# B&R Automation Studio project DuctLines (part 3)

### Program Logical/Feeder (IEC)

#### Cyclic.ld - Cyclic code
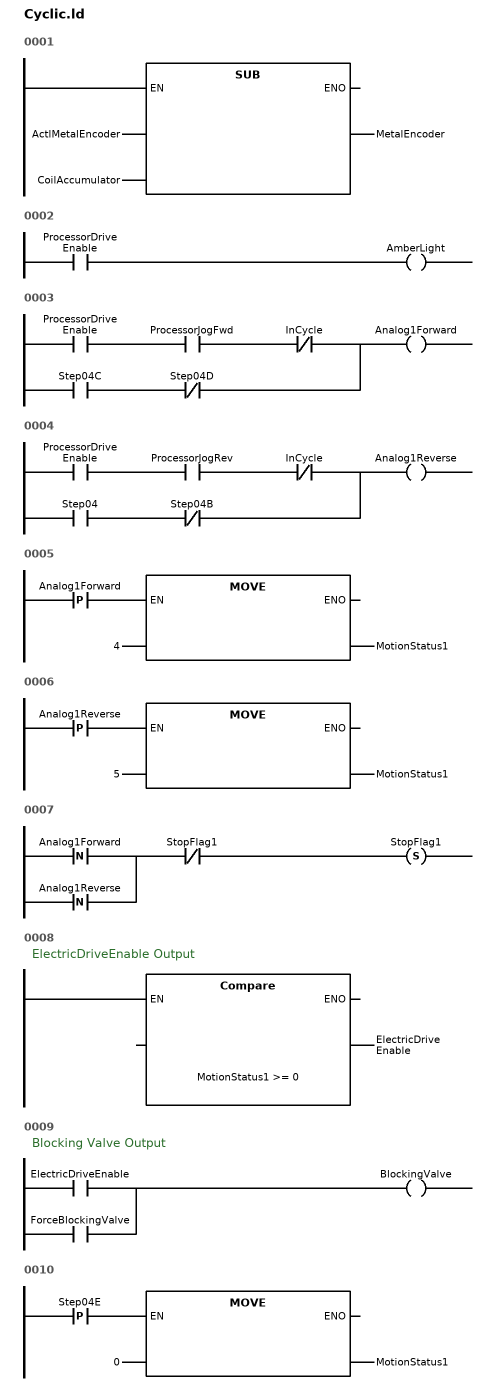
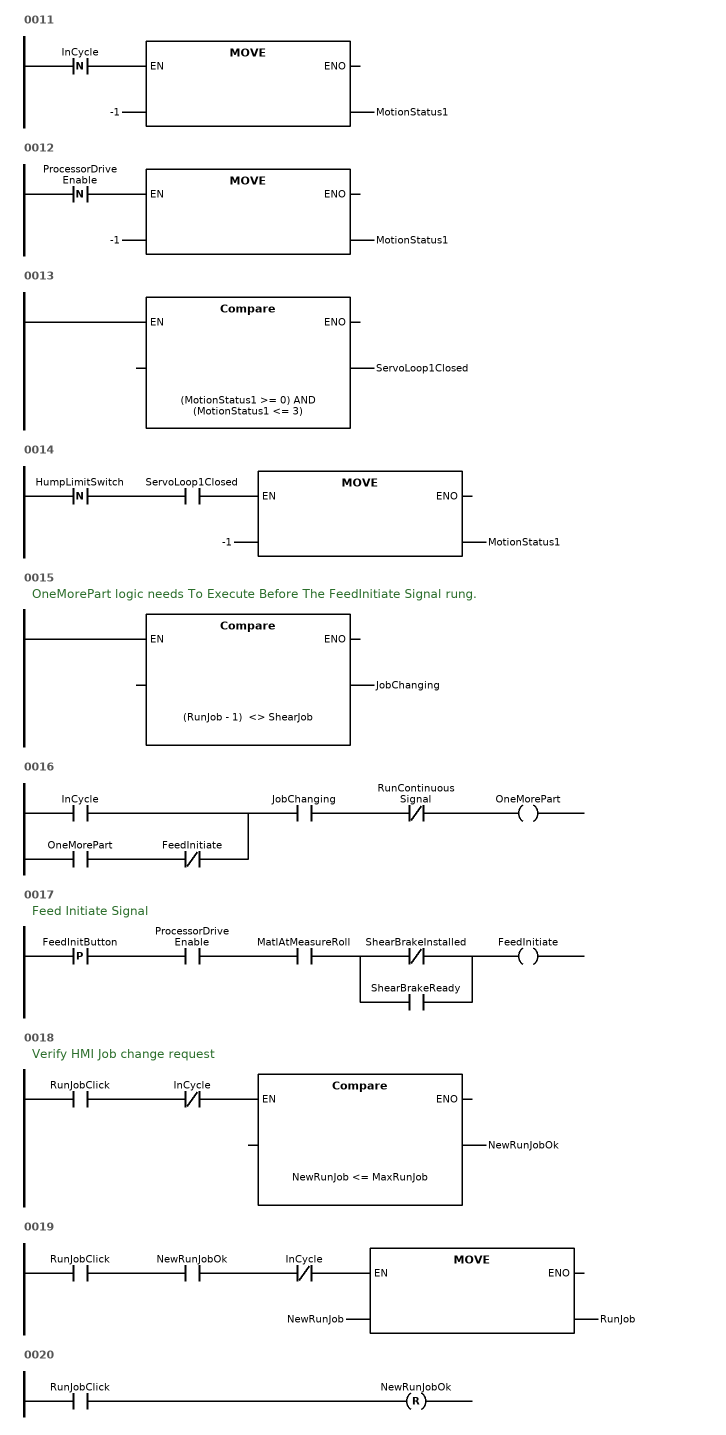
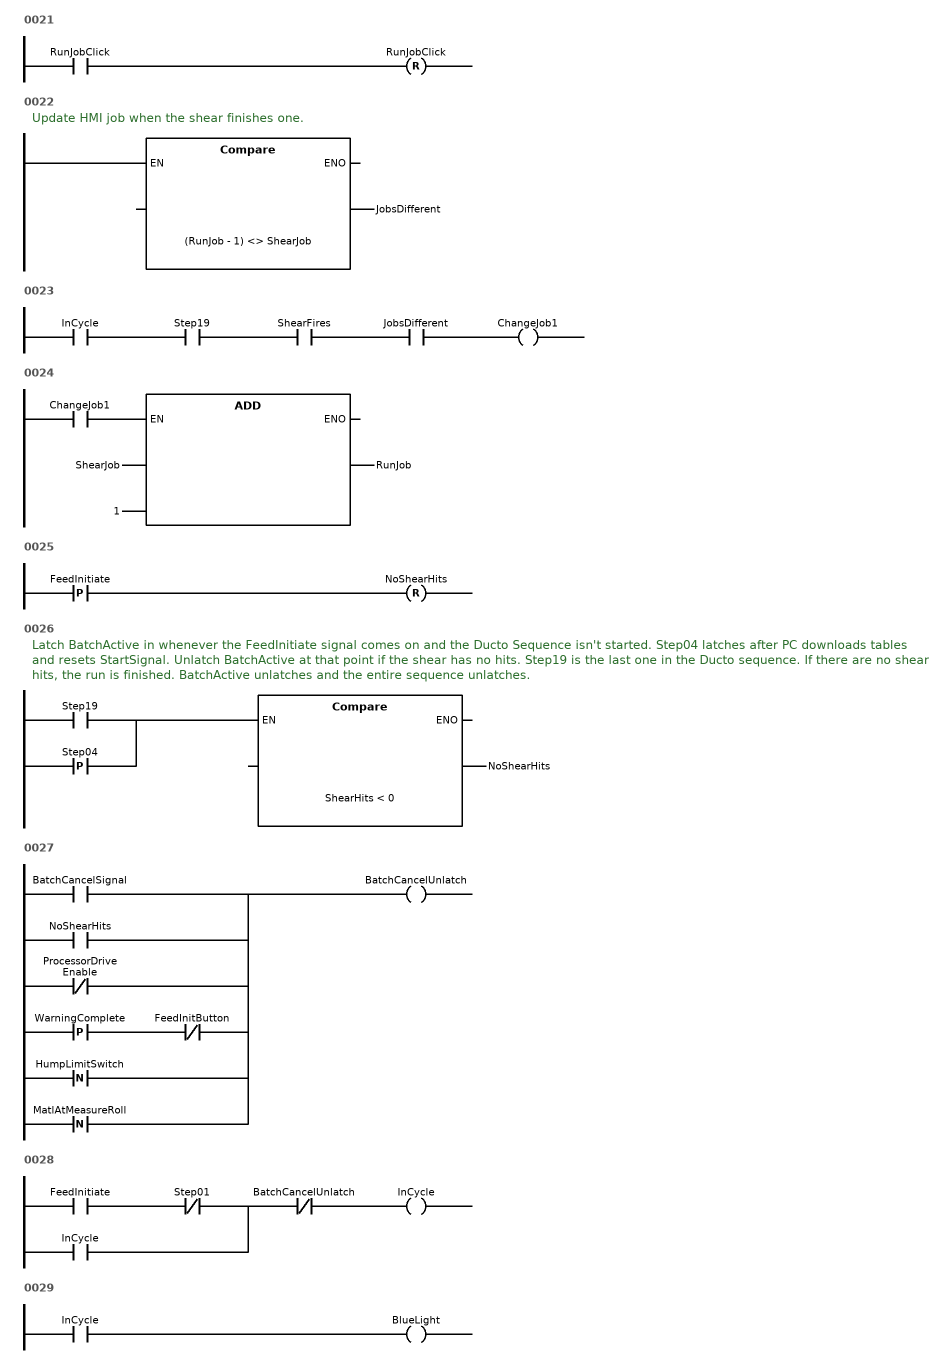
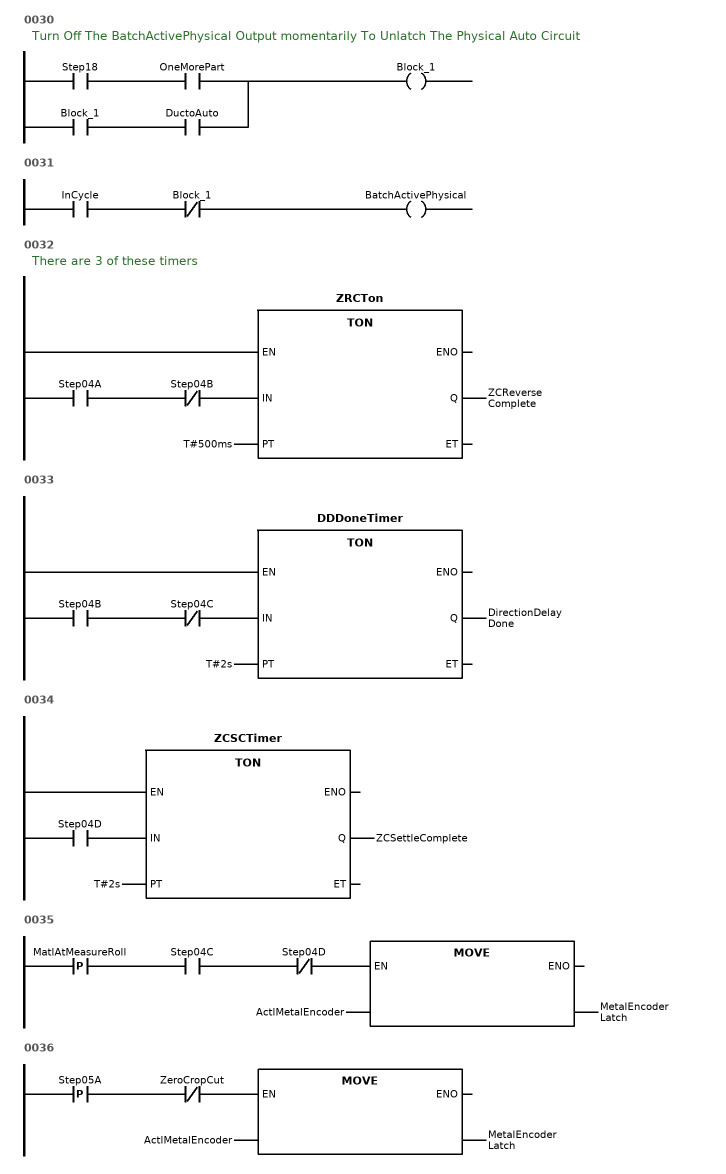
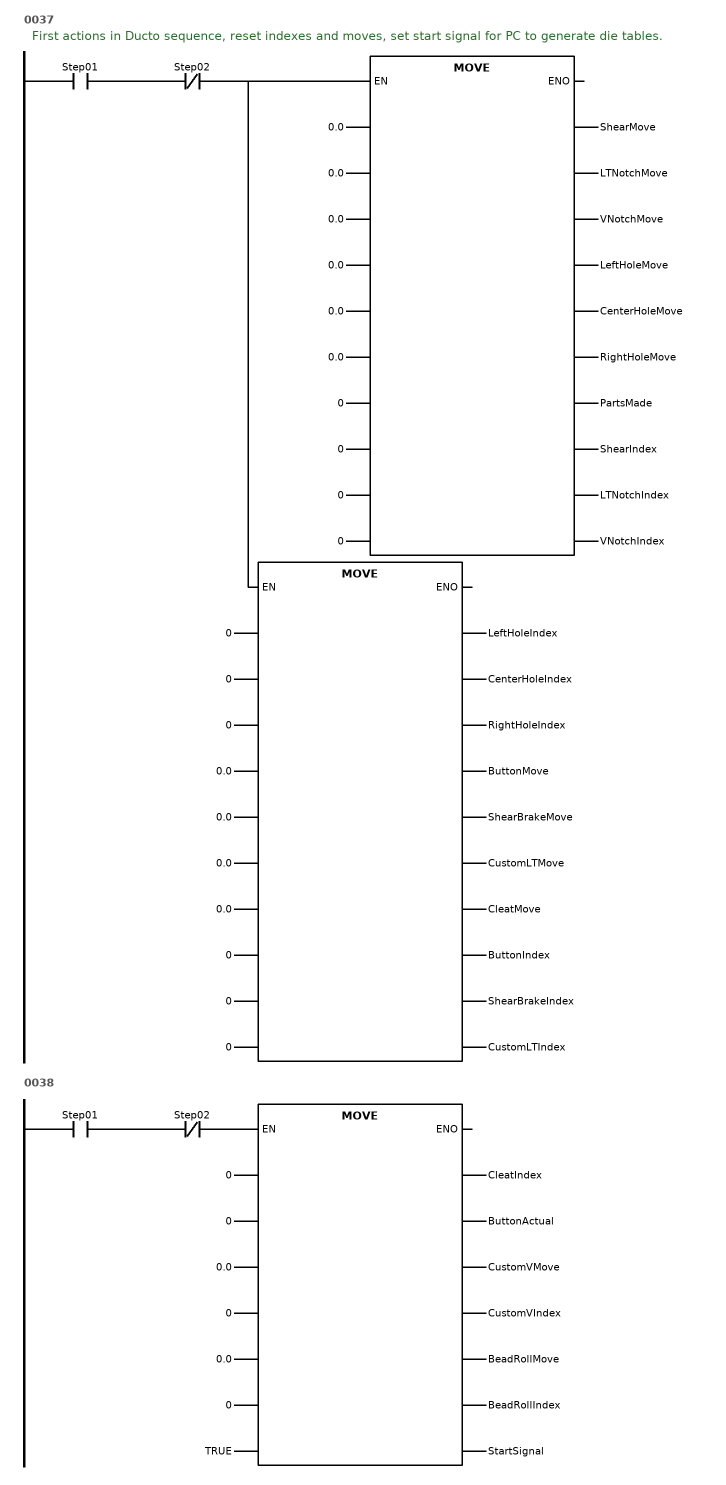
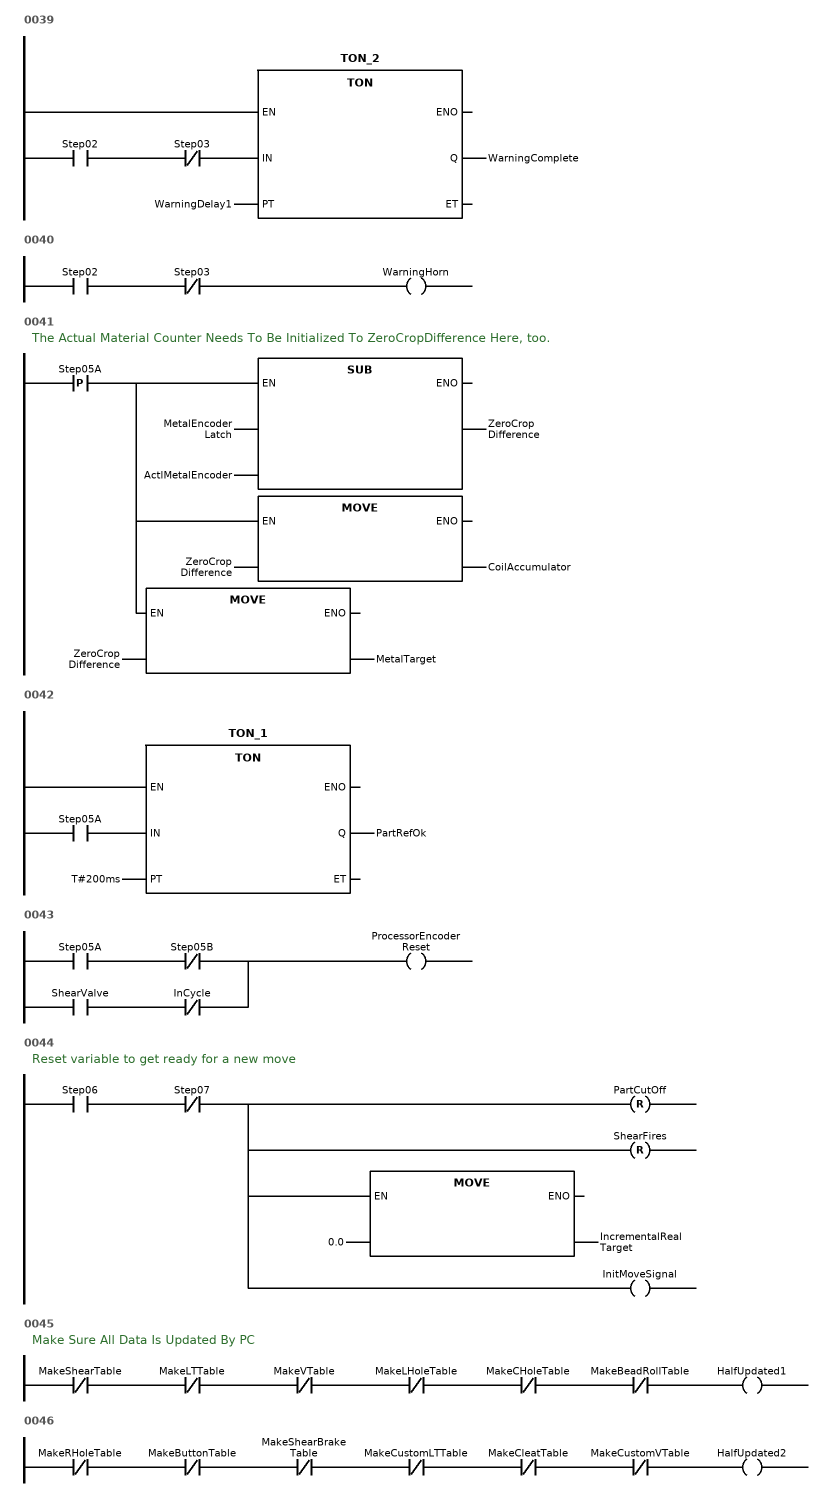
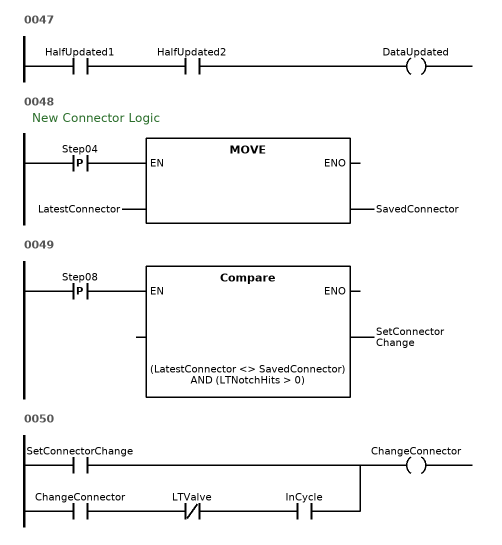
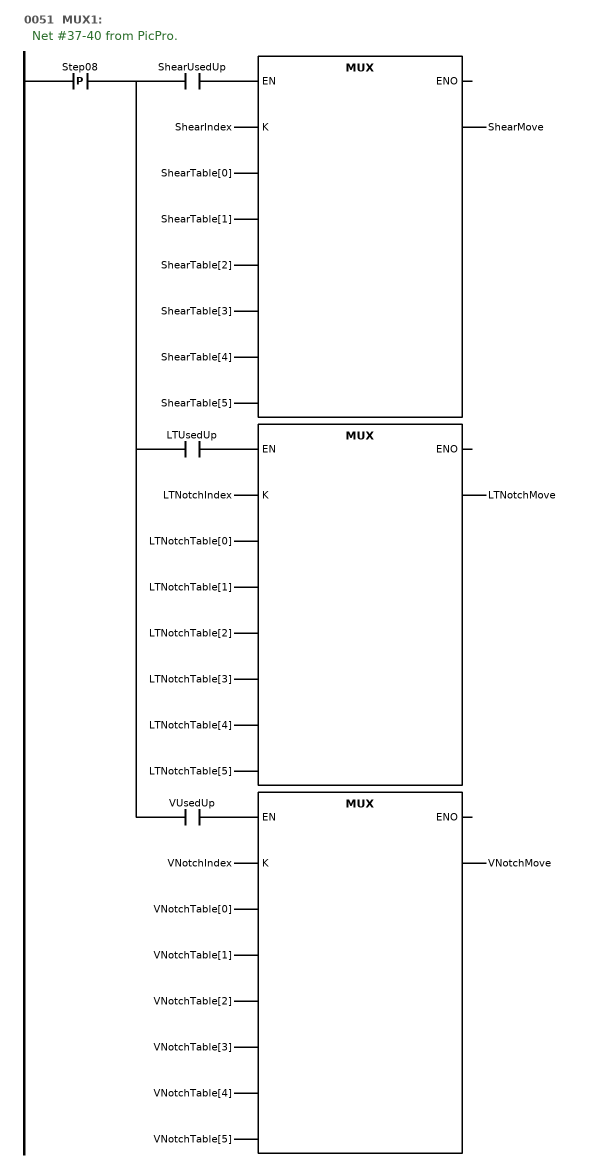
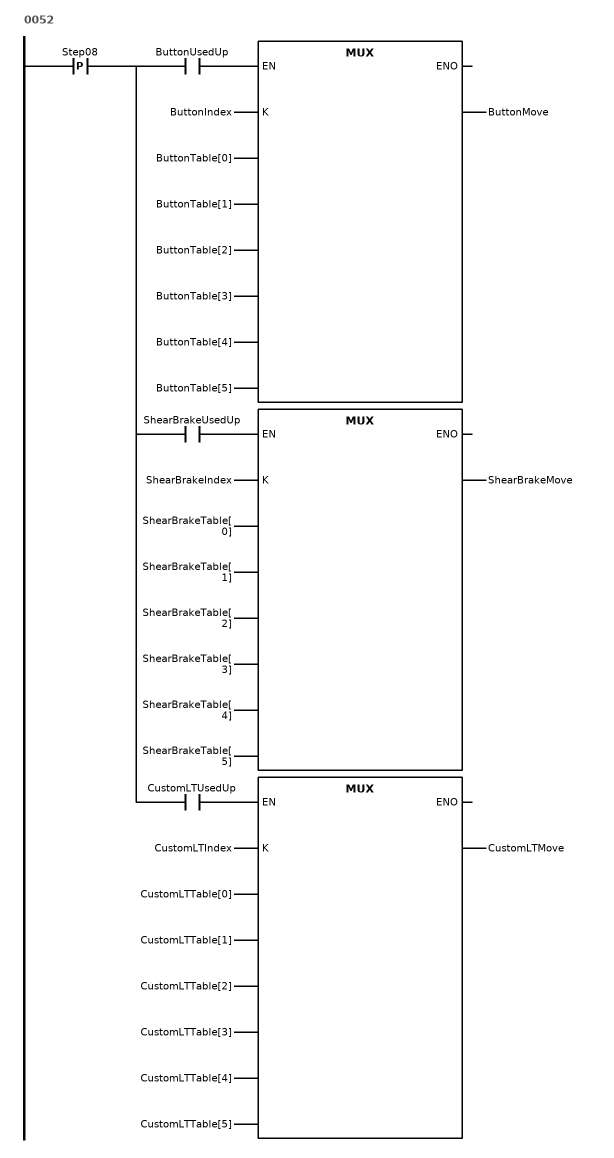
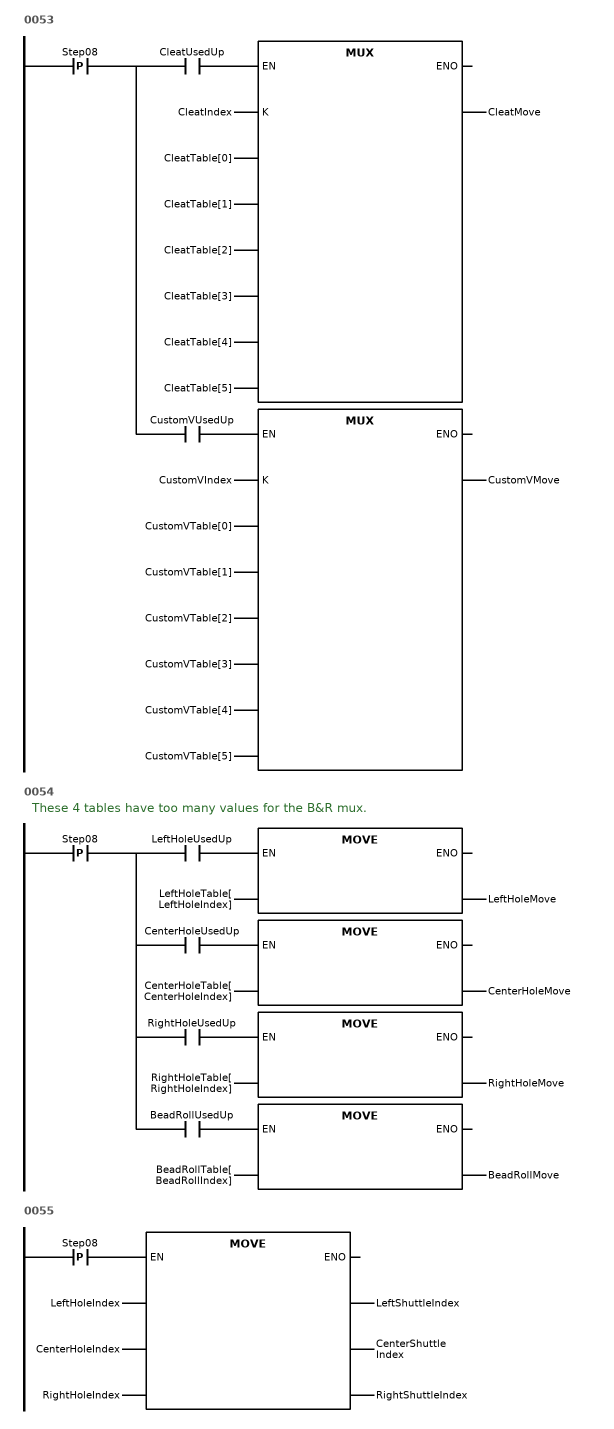
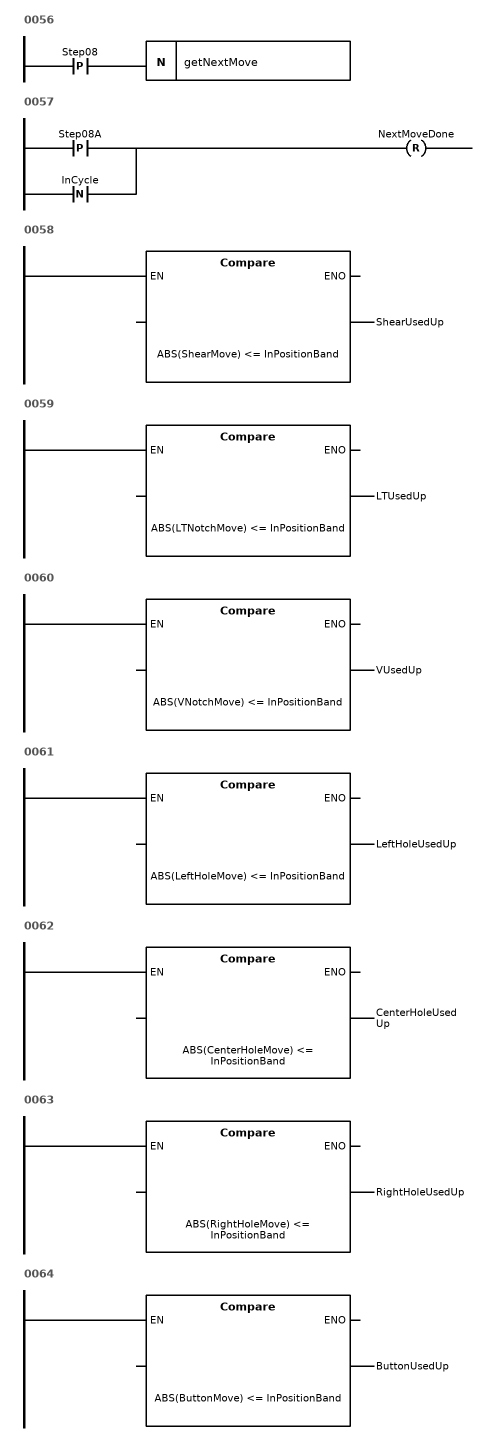
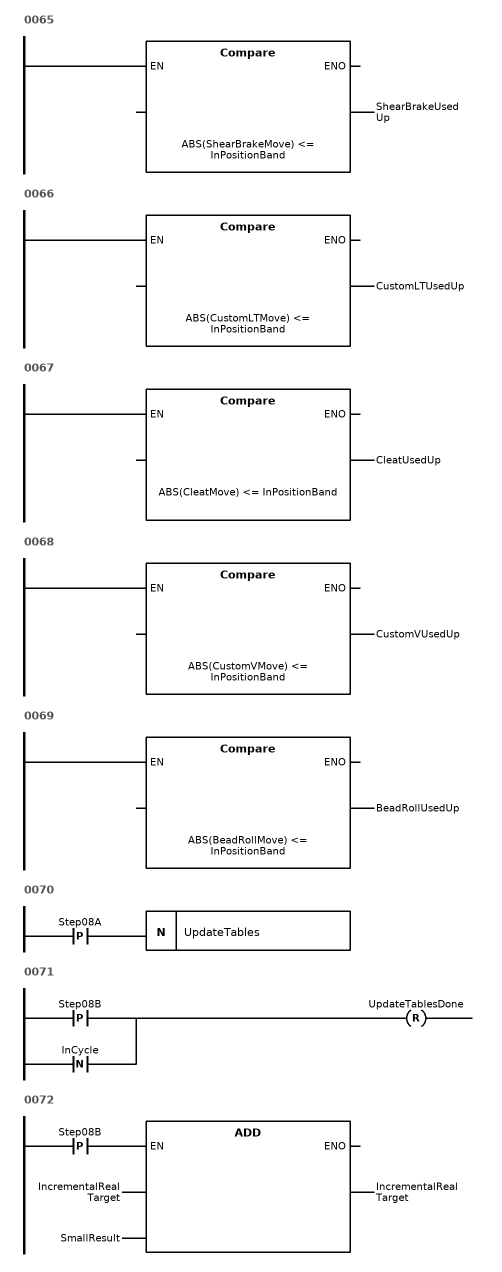
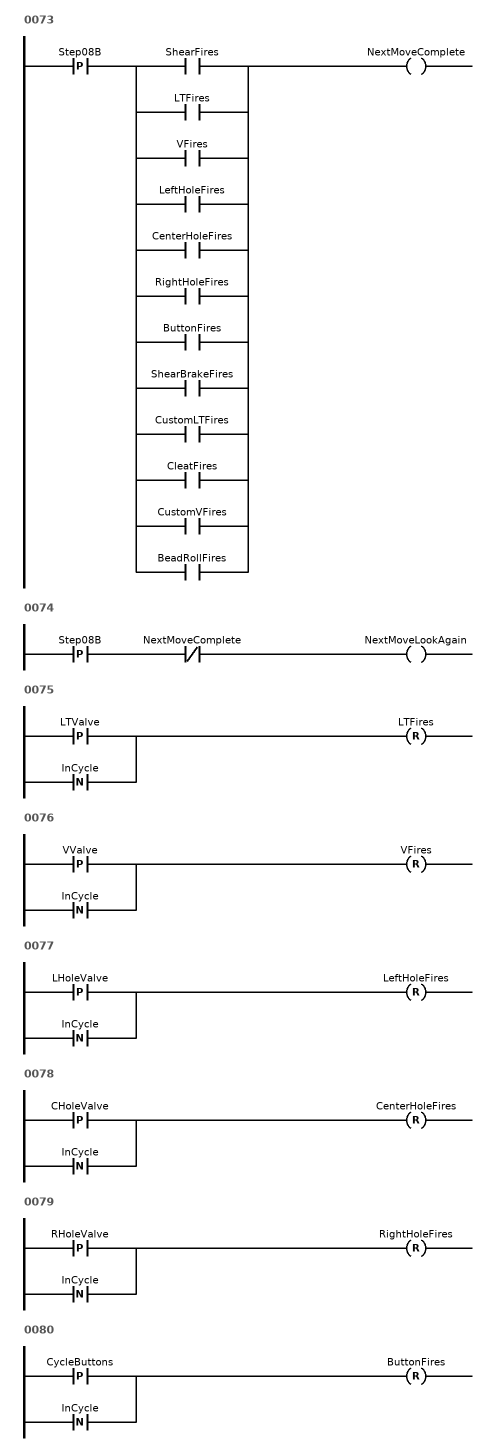
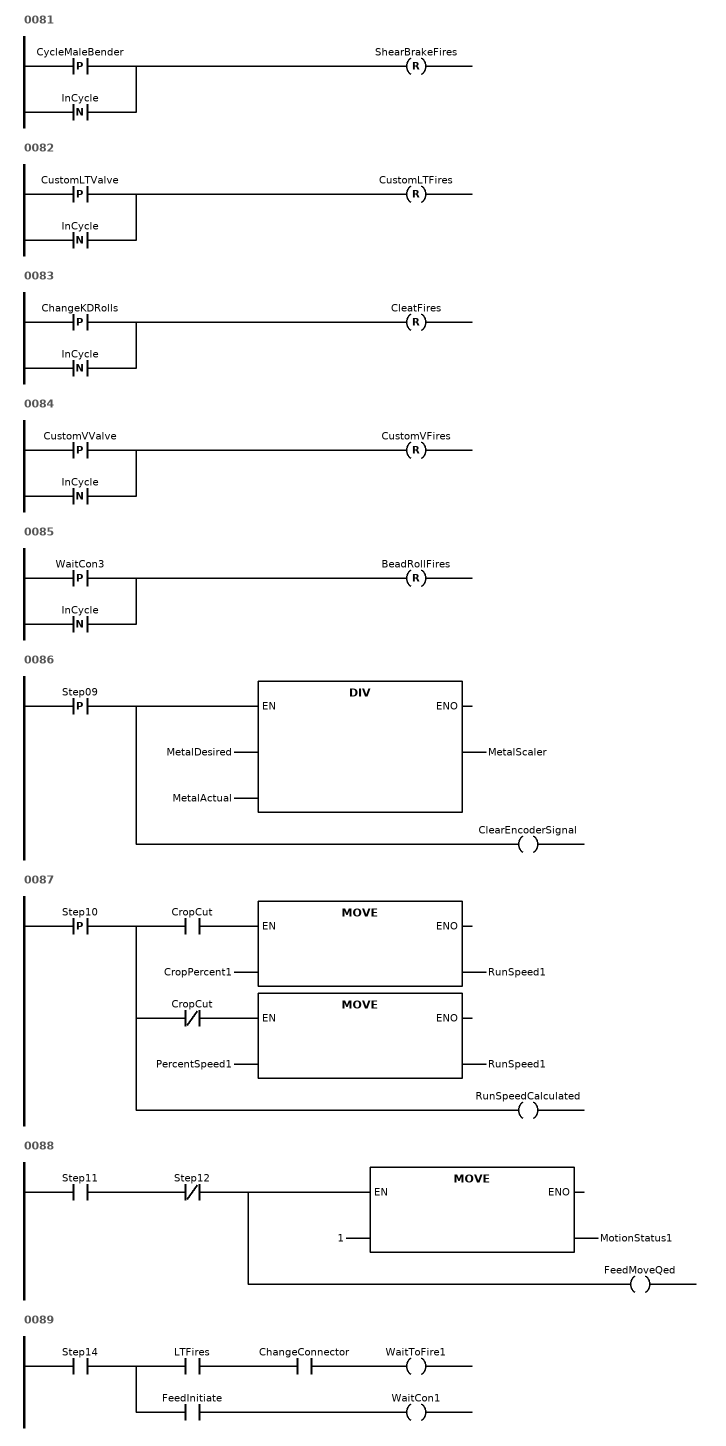
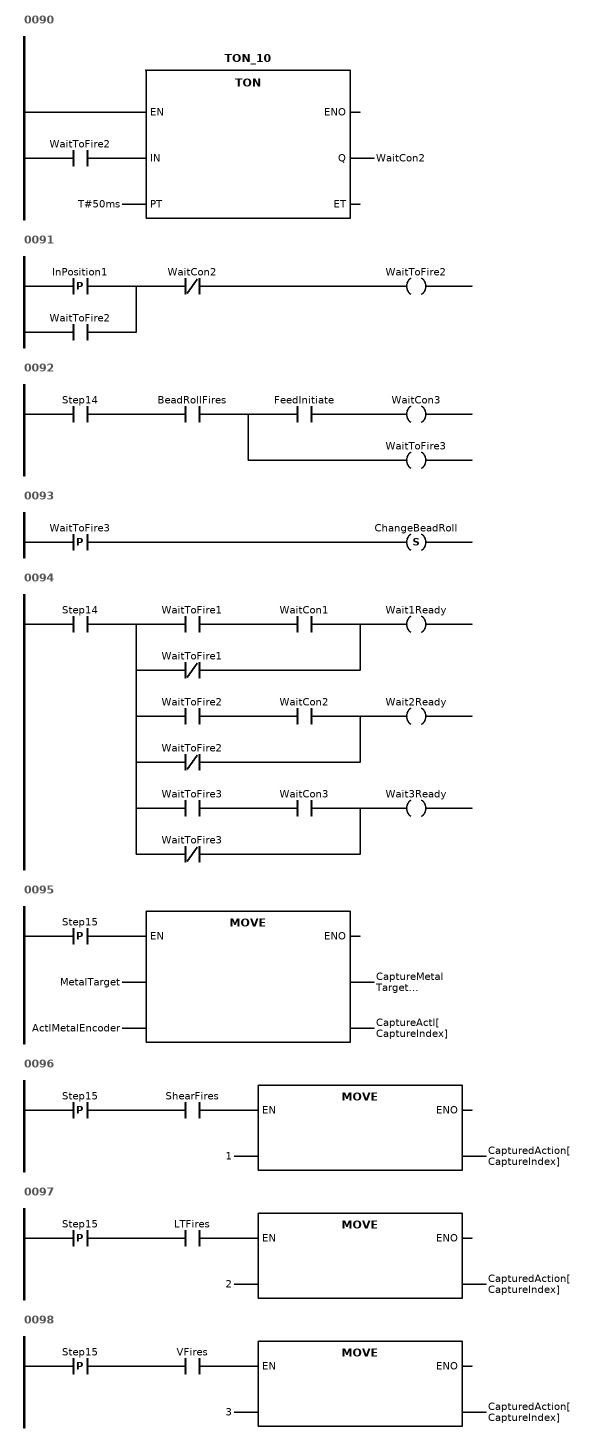
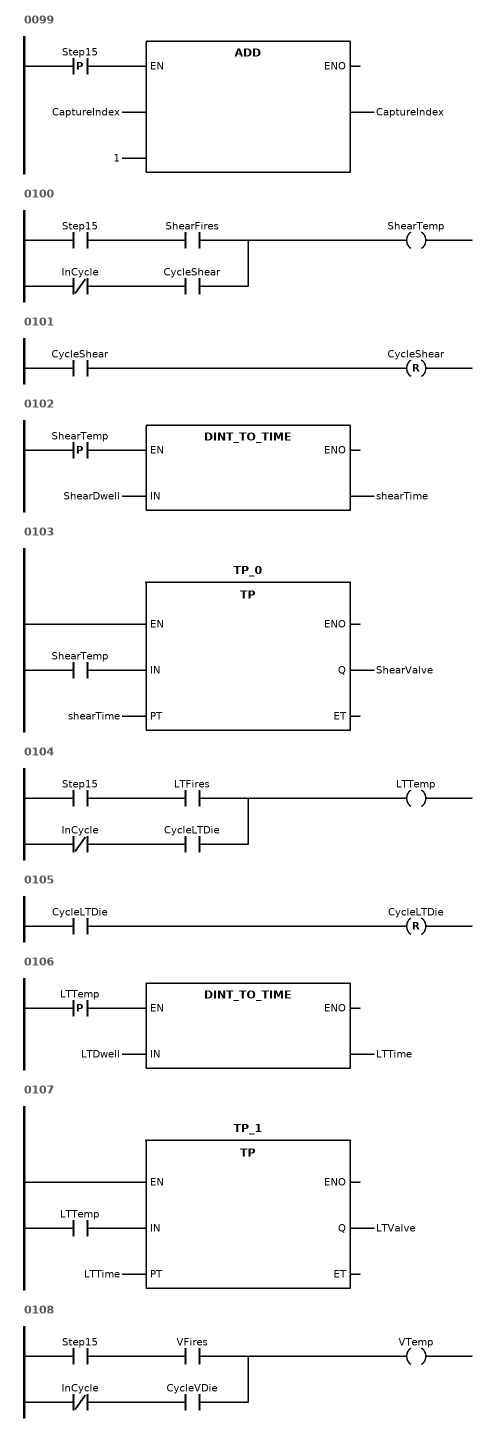
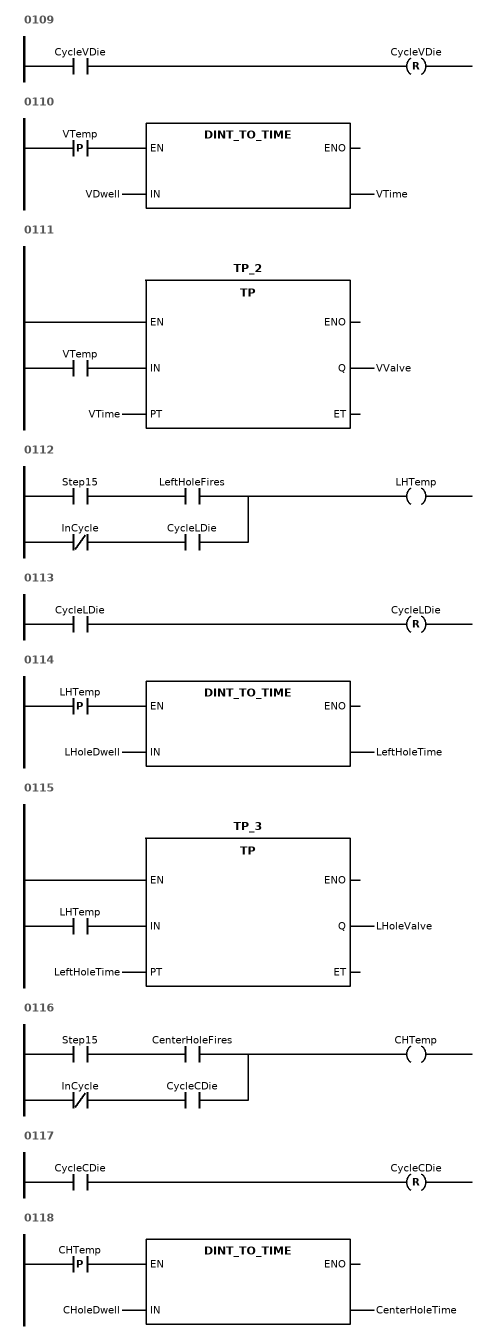
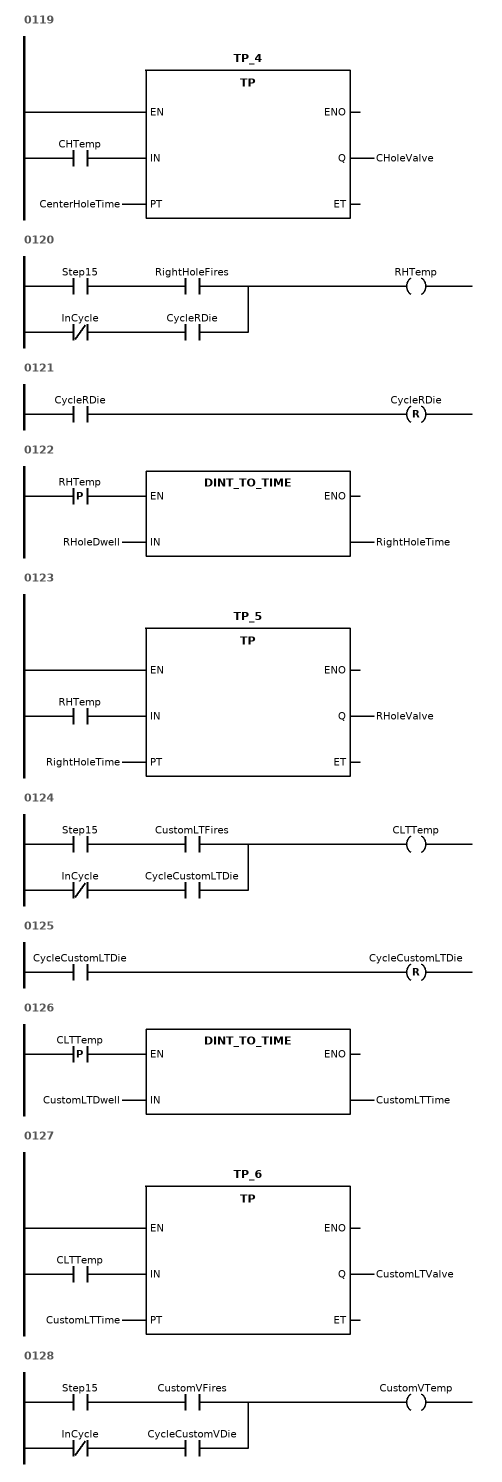
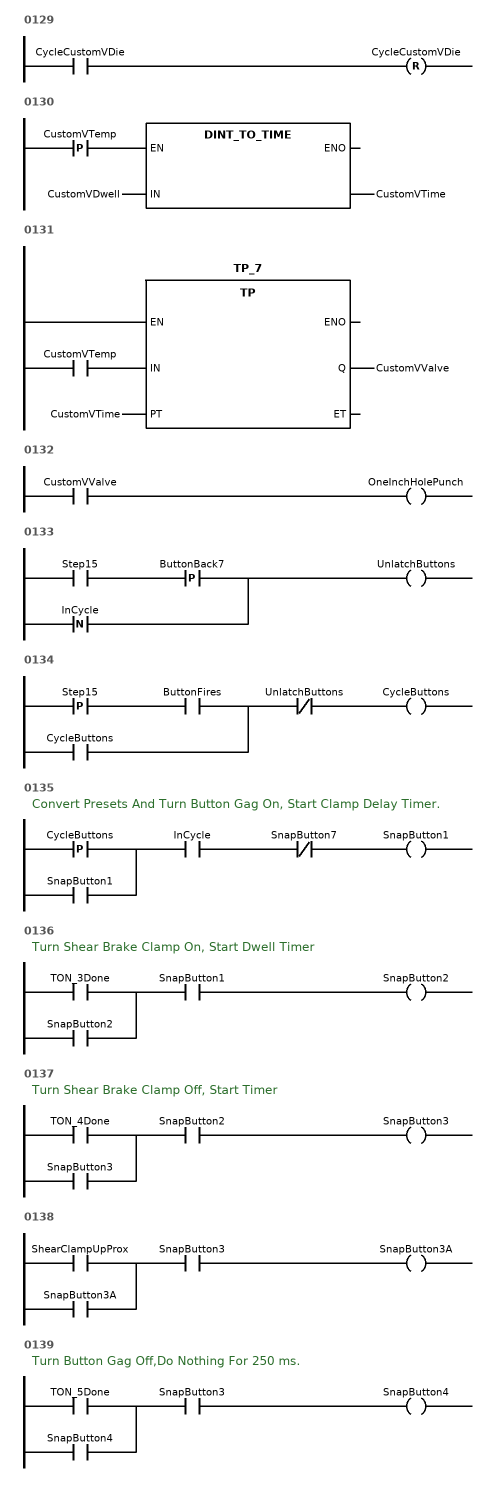
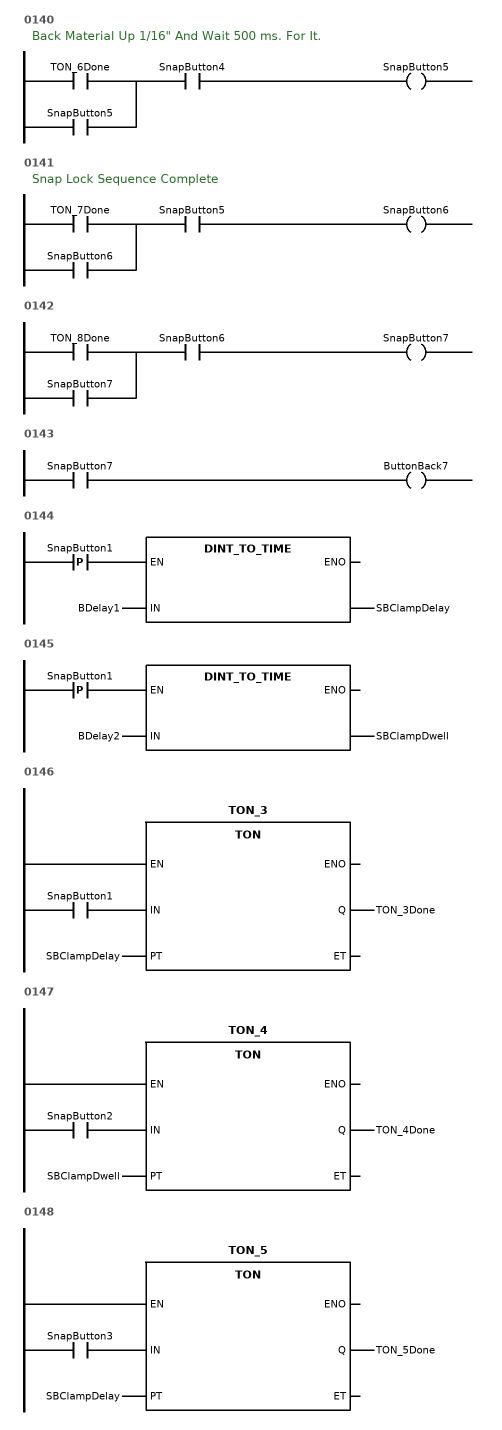
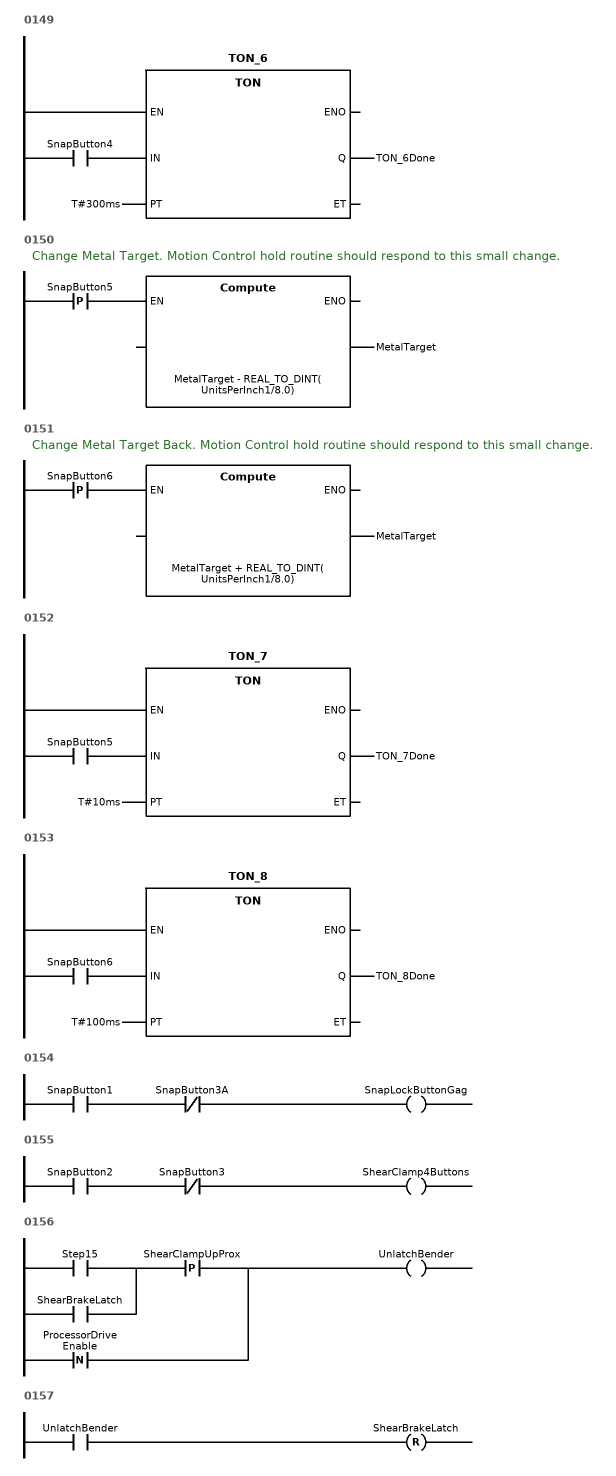
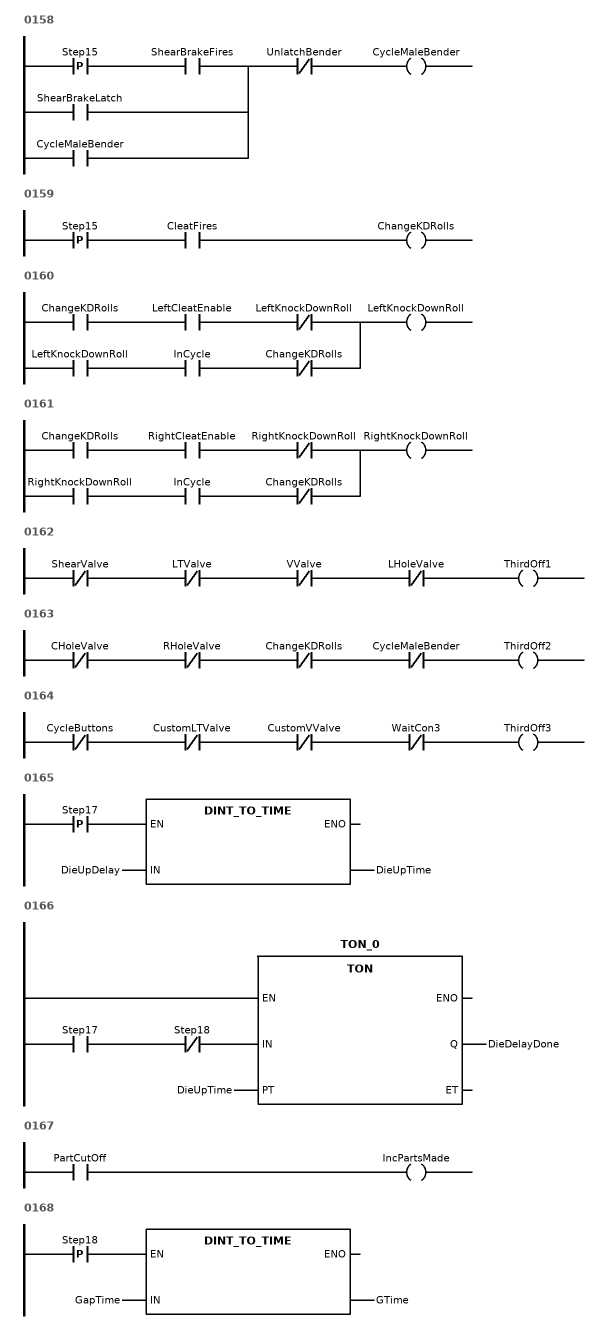
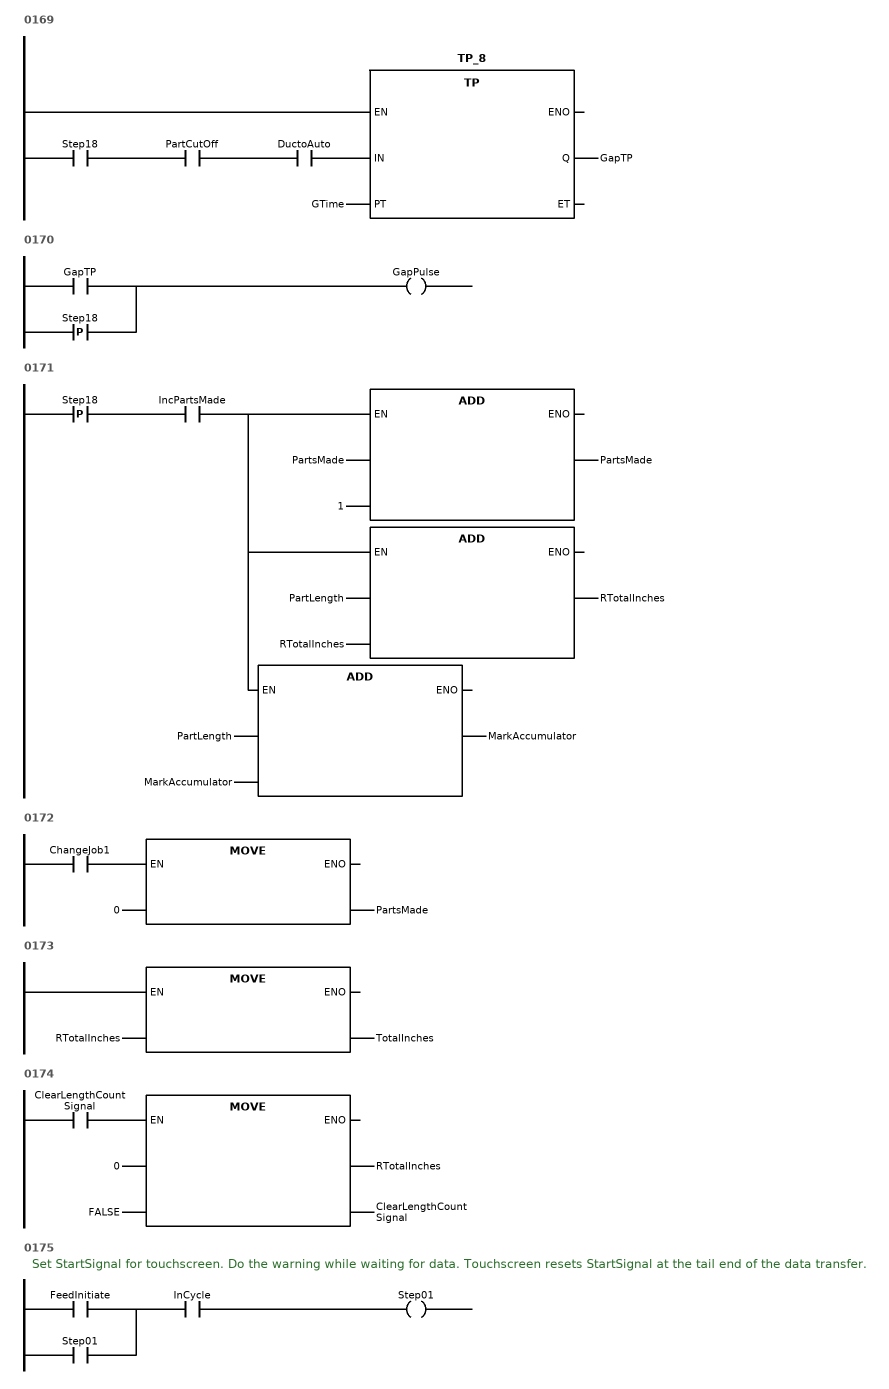
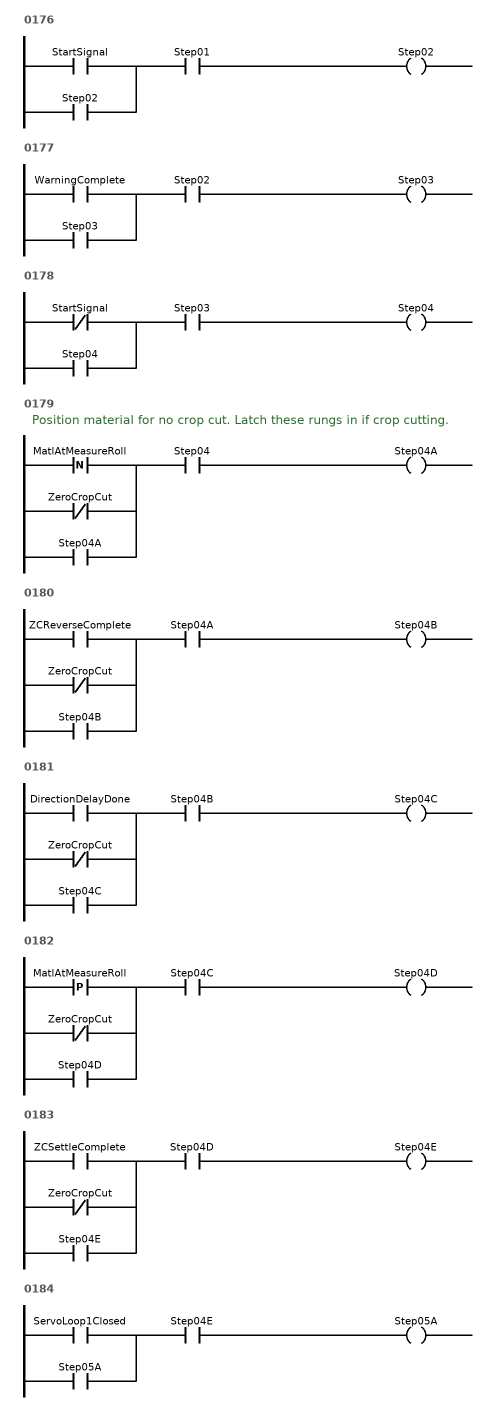
